(* IEC 61131-3 sources: CodesysTest/export/Unused/FB_SimBasicPrinter.pou/PrintDone.prop, 1 file *)

(* ---- Get.pm.st ---- *)
(*#-#-#-#-#-#-#-#-#-#---Declaration---#-#-#-#-#-#-#-#-#-#-#-#-#*)

VAR
END_VAR
(*#-#-#-#-#-#-#-#-#-#---Implementation---#-#-#-#-#-#-#-#-#-#-#-#-#*)

PrintDone := beginPrinting.Q;
